INTERFACE I_QuantityPublic EXTENDS I_Quantity, I_FalliblePublic


PROPERTY Units : T_MaxString
SET
END_SET
END_PROPERTY

END_INTERFACE

(* stored: Version 1.1.0.1
   Itf I_QuantityPublic: Id {a7793ee0-65b7-4394-ab1b-a37056379501}
   Property Units: Id {a6b68181-a638-46b2-8ae5-b31f49b43321}
   Set Set: Id {01d71d8e-f75c-4d0d-acf9-8caaede3e6d1} *)
